INTERFACE IPerson_Object EXTENDS TcoCore.ITcoObject

METHOD Accept : BOOL
VAR_INPUT
END_VAR
END_METHOD

METHOD Refuse : BOOL
VAR_INPUT
END_VAR
END_METHOD

METHOD PUBLIC RequestForFavor
VAR_INPUT
	inRequestedFavor	:	STRING;
	inReturnFavor		:	STRING;
END_VAR
END_METHOD

END_INTERFACE

(* stored: Version 1.1.0.1, ProductVersion 3.1.4024.6
   Itf IPerson_Object: Id {ad495d6f-6831-0e74-1e94-18ac17fa1c77}
   Method Accept: Id {9dbf19c4-a5e3-0af4-0444-a3098608e93d}
   Method Refuse: Id {1e28acde-074e-04f4-2cfa-8e25a152b64d}
   Method RequestForFavor: Id {9d333f29-8850-0eab-069a-14e73f68b7c9} *)
